// TIA Portal V20 export
DATA_BLOCK "InstCallEquipment"   // DB126
{ DB_Accessible_From_OPC_UA := 'FALSE' }
AUTHOR : ERsystem_FA2_DH. Kim
// stored: AssignedProDiagFB Unit1.Em3.ProDiag, DBAccessibleFromOPCUA false, DBAccessibleFromWebserver false, InstanceOfName Unit1.Em3.CallEquipment, InstanceOfType FB, Namespace Unit1.Em3
"Unit1.Em3.CallEquipment"
   // VAR_INPUT
   //    ZoneOperationEnable { ExternalWritable := 'False'} : "LWONIK_typeSafetyZoneManualOperation";
   // END_VAR
   // VAR_IN_OUT
   //    unitStatus : "LAF_typeUnitStatus";
   //    unitAlarmDB : "LAF_typeAlarms";
   //    emFeedback : "LUC_typeEmFeedback";
   // END_VAR
   // VAR
   //    InstSequenceWebGuide : "Unit1.Em3.Sequence_1_WebGuide";
   //    instWebGuideHomeJob1 { S7_SetPoint := 'True'} : "LAF_SelectJob";
   //    instWebGuideGuidingJob2 { S7_SetPoint := 'True'} : "LAF_SelectJob";
   //    instCmSafetyPinIdlePositionSensor : "LBC_DigitalSignalCn";
   //    instCmIonizerTopMaintDetection { S7_SetPoint := 'True'} : "LBC_DigitalSignalCn";
   //    instCmIonizerTopErrorDetection { S7_SetPoint := 'True'} : "LBC_DigitalSignalCn";
   //    instCmIonizerBtmMaintDetection { S7_SetPoint := 'True'} : "LBC_DigitalSignalCn";
   //    instCmIonizerBtmErrorDetection { S7_SetPoint := 'True'} : "LBC_DigitalSignalCn";
   //    instCmDancerEncoder { ExternalAccessible := 'False'; ExternalVisible := 'False'; ExternalWritable := 'False'; S7_SetPoint := 'True'} : "LBC_AnalogInputCn";
   //    instCmLoadCellControllerInterface { ExternalAccessible := 'False'; ExternalVisible := 'False'; ExternalWritable := 'False'; S7_SetPoint := 'True'} : "LBC_AnalogInputCn";
   //    instCmDancerElectroPneumaticRegulator { ExternalAccessible := 'False'; ExternalVisible := 'False'; ExternalWritable := 'False'; S7_SetPoint := 'True'} : "LBC_AnalogOutputCn";
   //    instCmCompensatorAxisX { S7_SetPoint := 'True'} : "LBC_Axis64Pos_TecPlcCn";
   //    instCmUnwinderVirtualAxisX { S7_SetPoint := 'True'} : "LBC_Axis64Pos_TecPlcCn";
   //    instInterlockCompensatorAxisX { S7_SetPoint := 'True'} : "LER_Axis64Pos_InterlockSummary";
   //    instInterlockUnwinderVirtualAxisX { S7_SetPoint := 'True'} : "LER_Axis64Pos_InterlockSummary";
   //    instCmDancerFwdBwd { ExternalAccessible := 'False'; ExternalVisible := 'False'; ExternalWritable := 'False'; S7_SetPoint := 'True'} : "LBC_TwoWayActuatorCn";
   //    instCmSepaUnwinderIonizerTop { ExternalAccessible := 'False'; ExternalVisible := 'False'; ExternalWritable := 'False'; S7_SetPoint := 'True'} : "LBC_TwoWayActuatorCn";
   //    instCmSepaUnwinderIonizerBottom { ExternalAccessible := 'False'; ExternalVisible := 'False'; ExternalWritable := 'False'; S7_SetPoint := 'True'} : "LBC_TwoWayActuatorCn";
   //    instCmEpcPivot { ExternalAccessible := 'False'; ExternalVisible := 'False'; ExternalWritable := 'False'; S7_SetPoint := 'True'} : "LER_EPC_CON600";
   //    instManageAlarms { ExternalWritable := 'False'} : "LAF_ManageAlarms";
   //    instEventsPFE : "Unit1.Em3.EventsPFE";
   //    statUnitStatus { ExternalWritable := 'False'} : "LAF_typeUnitStatus";
   //    statSlmStatus : Struct
   //       running { ExternalWritable := 'False'} : Bool;
   //       powerOff { ExternalWritable := 'False'} : Bool;
   //    END_STRUCT;
   //    statTonTime { ExternalAccessible := 'False'; ExternalVisible := 'False'; ExternalWritable := 'False'} : Array[0..1999] of TON_TIME;
   //    statTofTime { ExternalAccessible := 'False'; ExternalVisible := 'False'; ExternalWritable := 'False'} : Array[0..99] of TOF_TIME;
   //    statPulse { ExternalAccessible := 'False'; ExternalVisible := 'False'; ExternalWritable := 'False'} : Struct
   //       miscellaneous : Array[0..99] of Bool;
   //       workingDone : Struct
   //          mainPnP : Array[0..99] of Bool;
   //          alignTable : Array[0..99] of Bool;
   //          ngPnP : Array[0..99] of Bool;
   //       END_STRUCT;
   //       axisEnable : Array[0..99] of Bool;
   //       brakeTest : Array[0..99] of Bool;
   //    END_STRUCT;
   //    statEnableManualCmds : Bool := TRUE;
   //    Scan_on : Bool;
   //    "*** Interlock Axis ***" { ExternalAccessible := 'False'; ExternalVisible := 'False'; ExternalWritable := 'False'} : Bool;
   //    "compenastor X Home" { S7_SetPoint := 'True'} : "Homing.LER_Axis";
   //    "compenastor X Jog_CW" { S7_SetPoint := 'True'} : "Jog.LER_Axis";
   //    "compenastor X Jog_CCW" { S7_SetPoint := 'True'} : "Jog.LER_Axis";
   //    "compenastor X Position_" { S7_SetPoint := 'True'} : Array[0..5] of "Position.LER_Axis";
   //    "*** Interlock Actuator ******" { ExternalAccessible := 'False'; ExternalVisible := 'False'; ExternalWritable := 'False'} : Bool;
   //    "DancerFwdBwd Home" { S7_SetPoint := 'True'} : "Cylinder.LER_Actuator";
   //    "DancerFwdBwd Work" { S7_SetPoint := 'True'} : "Cylinder.LER_Actuator";
   //    "SepaUnwinderIonizer Home" { S7_SetPoint := 'True'} : "Cylinder.LER_Actuator";
   //    "SepaUnwinderIonizer Work" { S7_SetPoint := 'True'} : "Cylinder.LER_Actuator";
   //    "SepaUnwinderIonizerBottom Home" { S7_SetPoint := 'True'} : "Cylinder.LER_Actuator";
   //    "SepaUnwinderIonizerBottom Work" { S7_SetPoint := 'True'} : "Cylinder.LER_Actuator";
   //    AXIS3 : "LER_CM_Name";
   //    Cylinder10 : "LER_CM_Name";
   //    instCmRotaionSafetyPinPositionSensor { ExternalAccessible := 'False'; ExternalVisible := 'False'; ExternalWritable := 'False'} : "LBC_DigitalSignalCn";
   //    citi_Ptrig : Array[0..20] of Bool;
   //    citiTon : Array[0..20] of TON_TIME;
   //    citi : Time;
   //    citiTest : Array[0..20] of Bool;
   // END_VAR
BEGIN
   ZoneOperationEnable.autoStartEnable := FALSE;
   ZoneOperationEnable.doorLockEnable := TRUE;
   ZoneOperationEnable.doorUnlockEnable := TRUE;
   ZoneOperationEnable.rc_AutoEnable := FALSE;
   ZoneOperationEnable.rc_RollChangeEnable := FALSE;
   ZoneOperationEnable.rc_DoorLockEnable := TRUE;
   ZoneOperationEnable.rc_DoorUnlockEnable := TRUE;
   ZoneOperationEnable.hmiOperationEnable := TRUE;
   ZoneOperationEnable.phmiOperationEnable := FALSE;
   instCmSafetyPinIdlePositionSensor.enable := TRUE;
   instCmSafetyPinIdlePositionSensor.parentReferenceDesignator := WSTRING#'U1.EM3 WebGuide';
   instCmSafetyPinIdlePositionSensor.digitalValue := TRUE;
   instCmSafetyPinIdlePositionSensor.simulatedDigitalValue := FALSE;
   instCmSafetyPinIdlePositionSensor.statProcessValues.enable := TRUE;
   instCmSafetyPinIdlePositionSensor.statProcessValues.referenceDesignator := WSTRING#'U1.EM3 WebGuide.DigitalSignal';
   instCmSafetyPinIdlePositionSensor.statProcessValues.simulation := FALSE;
   instCmSafetyPinIdlePositionSensor.statProcessValues.processValue := TRUE;
   instCmSafetyPinIdlePositionSensor.statProcessValues.error := FALSE;
   instCmSafetyPinIdlePositionSensor.statProcessValues.status := 16#0000;
   instCmSafetyPinIdlePositionSensor.statDiagnostics.status := 16#0000;
   instCmSafetyPinIdlePositionSensor.statDiagnostics.subfunctionStatus := 16#0000;
   instCmSafetyPinIdlePositionSensor.statDiagnostics.stateNumber := 0;
   instCmSafetyPinIdlePositionSensor.statEmptyDiagnostics.status := 16#0000;
   instCmSafetyPinIdlePositionSensor.statEmptyDiagnostics.subfunctionStatus := 16#0000;
   instCmSafetyPinIdlePositionSensor.statEmptyDiagnostics.stateNumber := 0;
   instCmSafetyPinIdlePositionSensor.instOnDelay.PT := T#0MS;
   instCmSafetyPinIdlePositionSensor.instOnDelay.IN := FALSE;
   instCmSafetyPinIdlePositionSensor.instOffDelay.PT := T#0MS;
   instCmSafetyPinIdlePositionSensor.instOffDelay.IN := FALSE;
   instCmSafetyPinIdlePositionSensor.statDisableAlarms := FALSE;
   instCmSafetyPinIdlePositionSensor.statErrorState := 16#0000;
   instCmSafetyPinIdlePositionSensor.statFirstCall := FALSE;
   instCmSafetyPinIdlePositionSensor.statResetPrevious := FALSE;
   instCmSafetyPinIdlePositionSensor.statEnablePrevious := TRUE;
   instCmSafetyPinIdlePositionSensor.statProcessValuePrevious := TRUE;
   instCmIonizerTopMaintDetection.enable := TRUE;
   instCmIonizerTopMaintDetection.parentReferenceDesignator := WSTRING#'U1.EM3 WebGuide';
   instCmIonizerTopMaintDetection.digitalValue := FALSE;
   instCmIonizerTopMaintDetection.simulatedDigitalValue := FALSE;
   instCmIonizerTopMaintDetection.statProcessValues.enable := TRUE;
   instCmIonizerTopMaintDetection.statProcessValues.referenceDesignator := WSTRING#'U1.EM3 WebGuide.DigitalSignal';
   instCmIonizerTopMaintDetection.statProcessValues.simulation := FALSE;
   instCmIonizerTopMaintDetection.statProcessValues.processValue := FALSE;
   instCmIonizerTopMaintDetection.statProcessValues.error := FALSE;
   instCmIonizerTopMaintDetection.statProcessValues.status := 16#0000;
   instCmIonizerTopMaintDetection.statDiagnostics.status := 16#0000;
   instCmIonizerTopMaintDetection.statDiagnostics.subfunctionStatus := 16#0000;
   instCmIonizerTopMaintDetection.statDiagnostics.stateNumber := 0;
   instCmIonizerTopMaintDetection.statEmptyDiagnostics.status := 16#0000;
   instCmIonizerTopMaintDetection.statEmptyDiagnostics.subfunctionStatus := 16#0000;
   instCmIonizerTopMaintDetection.statEmptyDiagnostics.stateNumber := 0;
   instCmIonizerTopMaintDetection.instOnDelay.PT := T#0MS;
   instCmIonizerTopMaintDetection.instOnDelay.IN := FALSE;
   instCmIonizerTopMaintDetection.instOffDelay.PT := T#0MS;
   instCmIonizerTopMaintDetection.instOffDelay.IN := FALSE;
   instCmIonizerTopMaintDetection.statDisableAlarms := FALSE;
   instCmIonizerTopMaintDetection.statErrorState := 16#0000;
   instCmIonizerTopMaintDetection.statFirstCall := FALSE;
   instCmIonizerTopMaintDetection.statResetPrevious := FALSE;
   instCmIonizerTopMaintDetection.statEnablePrevious := TRUE;
   instCmIonizerTopMaintDetection.statProcessValuePrevious := FALSE;
   instCmIonizerTopErrorDetection.enable := TRUE;
   instCmIonizerTopErrorDetection.parentReferenceDesignator := WSTRING#'U1.EM3 WebGuide';
   instCmIonizerTopErrorDetection.digitalValue := TRUE;
   instCmIonizerTopErrorDetection.simulatedDigitalValue := FALSE;
   instCmIonizerTopErrorDetection.statProcessValues.enable := TRUE;
   instCmIonizerTopErrorDetection.statProcessValues.referenceDesignator := WSTRING#'U1.EM3 WebGuide.DigitalSignal';
   instCmIonizerTopErrorDetection.statProcessValues.simulation := FALSE;
   instCmIonizerTopErrorDetection.statProcessValues.processValue := TRUE;
   instCmIonizerTopErrorDetection.statProcessValues.error := FALSE;
   instCmIonizerTopErrorDetection.statProcessValues.status := 16#0000;
   instCmIonizerTopErrorDetection.statDiagnostics.status := 16#0000;
   instCmIonizerTopErrorDetection.statDiagnostics.subfunctionStatus := 16#0000;
   instCmIonizerTopErrorDetection.statDiagnostics.stateNumber := 0;
   instCmIonizerTopErrorDetection.statEmptyDiagnostics.status := 16#0000;
   instCmIonizerTopErrorDetection.statEmptyDiagnostics.subfunctionStatus := 16#0000;
   instCmIonizerTopErrorDetection.statEmptyDiagnostics.stateNumber := 0;
   instCmIonizerTopErrorDetection.instOnDelay.PT := T#0MS;
   instCmIonizerTopErrorDetection.instOnDelay.IN := FALSE;
   instCmIonizerTopErrorDetection.instOffDelay.PT := T#0MS;
   instCmIonizerTopErrorDetection.instOffDelay.IN := FALSE;
   instCmIonizerTopErrorDetection.statDisableAlarms := FALSE;
   instCmIonizerTopErrorDetection.statErrorState := 16#0000;
   instCmIonizerTopErrorDetection.statFirstCall := FALSE;
   instCmIonizerTopErrorDetection.statResetPrevious := FALSE;
   instCmIonizerTopErrorDetection.statEnablePrevious := TRUE;
   instCmIonizerTopErrorDetection.statProcessValuePrevious := TRUE;
   instCmIonizerBtmMaintDetection.enable := TRUE;
   instCmIonizerBtmMaintDetection.parentReferenceDesignator := WSTRING#'U1.EM3 WebGuide';
   instCmIonizerBtmMaintDetection.digitalValue := FALSE;
   instCmIonizerBtmMaintDetection.simulatedDigitalValue := FALSE;
   instCmIonizerBtmMaintDetection.statProcessValues.enable := TRUE;
   instCmIonizerBtmMaintDetection.statProcessValues.referenceDesignator := WSTRING#'U1.EM3 WebGuide.DigitalSignal';
   instCmIonizerBtmMaintDetection.statProcessValues.simulation := FALSE;
   instCmIonizerBtmMaintDetection.statProcessValues.processValue := FALSE;
   instCmIonizerBtmMaintDetection.statProcessValues.error := FALSE;
   instCmIonizerBtmMaintDetection.statProcessValues.status := 16#0000;
   instCmIonizerBtmMaintDetection.statDiagnostics.status := 16#0000;
   instCmIonizerBtmMaintDetection.statDiagnostics.subfunctionStatus := 16#0000;
   instCmIonizerBtmMaintDetection.statDiagnostics.stateNumber := 0;
   instCmIonizerBtmMaintDetection.statEmptyDiagnostics.status := 16#0000;
   instCmIonizerBtmMaintDetection.statEmptyDiagnostics.subfunctionStatus := 16#0000;
   instCmIonizerBtmMaintDetection.statEmptyDiagnostics.stateNumber := 0;
   instCmIonizerBtmMaintDetection.instOnDelay.PT := T#0MS;
   instCmIonizerBtmMaintDetection.instOnDelay.IN := FALSE;
   instCmIonizerBtmMaintDetection.instOffDelay.PT := T#0MS;
   instCmIonizerBtmMaintDetection.instOffDelay.IN := FALSE;
   instCmIonizerBtmMaintDetection.statDisableAlarms := FALSE;
   instCmIonizerBtmMaintDetection.statErrorState := 16#0000;
   instCmIonizerBtmMaintDetection.statFirstCall := FALSE;
   instCmIonizerBtmMaintDetection.statResetPrevious := FALSE;
   instCmIonizerBtmMaintDetection.statEnablePrevious := TRUE;
   instCmIonizerBtmMaintDetection.statProcessValuePrevious := FALSE;
   instCmIonizerBtmErrorDetection.enable := TRUE;
   instCmIonizerBtmErrorDetection.parentReferenceDesignator := WSTRING#'U1.EM3 WebGuide';
   instCmIonizerBtmErrorDetection.digitalValue := TRUE;
   instCmIonizerBtmErrorDetection.simulatedDigitalValue := FALSE;
   instCmIonizerBtmErrorDetection.statProcessValues.enable := TRUE;
   instCmIonizerBtmErrorDetection.statProcessValues.referenceDesignator := WSTRING#'U1.EM3 WebGuide.DigitalSignal';
   instCmIonizerBtmErrorDetection.statProcessValues.simulation := FALSE;
   instCmIonizerBtmErrorDetection.statProcessValues.processValue := TRUE;
   instCmIonizerBtmErrorDetection.statProcessValues.error := FALSE;
   instCmIonizerBtmErrorDetection.statProcessValues.status := 16#0000;
   instCmIonizerBtmErrorDetection.statDiagnostics.status := 16#0000;
   instCmIonizerBtmErrorDetection.statDiagnostics.subfunctionStatus := 16#0000;
   instCmIonizerBtmErrorDetection.statDiagnostics.stateNumber := 0;
   instCmIonizerBtmErrorDetection.statEmptyDiagnostics.status := 16#0000;
   instCmIonizerBtmErrorDetection.statEmptyDiagnostics.subfunctionStatus := 16#0000;
   instCmIonizerBtmErrorDetection.statEmptyDiagnostics.stateNumber := 0;
   instCmIonizerBtmErrorDetection.instOnDelay.PT := T#0MS;
   instCmIonizerBtmErrorDetection.instOnDelay.IN := FALSE;
   instCmIonizerBtmErrorDetection.instOffDelay.PT := T#0MS;
   instCmIonizerBtmErrorDetection.instOffDelay.IN := FALSE;
   instCmIonizerBtmErrorDetection.statDisableAlarms := FALSE;
   instCmIonizerBtmErrorDetection.statErrorState := 16#0000;
   instCmIonizerBtmErrorDetection.statFirstCall := FALSE;
   instCmIonizerBtmErrorDetection.statResetPrevious := FALSE;
   instCmIonizerBtmErrorDetection.statEnablePrevious := TRUE;
   instCmIonizerBtmErrorDetection.statProcessValuePrevious := TRUE;
   instCmDancerEncoder.enable := TRUE;
   instCmDancerEncoder.parentReferenceDesignator := WSTRING#'U1.EM3 WebGuide';
   instCmDancerEncoder.analogValue := 13938;
   instCmDancerEncoder.simulatedAnalogValue := 0;
   instCmDancerEncoder.statProcessValues.enable := TRUE;
   instCmDancerEncoder.statProcessValues.referenceDesignator := WSTRING#'U1.EM3 WebGuide.cmDancerEncoder';
   instCmDancerEncoder.statProcessValues.simulation := FALSE;
   instCmDancerEncoder.statProcessValues.processValue := 0.354600694444443;
   instCmDancerEncoder.statProcessValues.analogValue := 13879;
   instCmDancerEncoder.statProcessValues.limitHigh2 := FALSE;
   instCmDancerEncoder.statProcessValues.limitHigh1 := FALSE;
   instCmDancerEncoder.statProcessValues.limitLow1 := FALSE;
   instCmDancerEncoder.statProcessValues.limitLow2 := FALSE;
   instCmDancerEncoder.statProcessValues.maxValueReached := FALSE;
   instCmDancerEncoder.statProcessValues.minValueReached := FALSE;
   instCmDancerEncoder.statProcessValues.error := FALSE;
   instCmDancerEncoder.statProcessValues.status := 16#0000;
   instCmDancerEncoder.statDiagnostics.status := 16#0000;
   instCmDancerEncoder.statDiagnostics.subfunctionStatus := 16#0000;
   instCmDancerEncoder.statDiagnostics.stateNumber := 0;
   instCmDancerEncoder.statEmptyDiagnostics.status := 16#0000;
   instCmDancerEncoder.statEmptyDiagnostics.subfunctionStatus := 16#0000;
   instCmDancerEncoder.statEmptyDiagnostics.stateNumber := 0;
   instCmDancerEncoder.statLimitationMessage := '';
   instCmDancerEncoder.statLimitMessage := '';
   instCmDancerEncoder.statErrorState := 16#0000;
   instCmDancerEncoder.statFirstCall := FALSE;
   instCmDancerEncoder.statDisableAlarms := FALSE;
   instCmDancerEncoder.statResetPrevious := FALSE;
   instCmDancerEncoder.statEnablePrevious := TRUE;
   instCmLoadCellControllerInterface.enable := TRUE;
   instCmLoadCellControllerInterface.parentReferenceDesignator := WSTRING#'U1.EM3 WebGuide';
   instCmLoadCellControllerInterface.analogValue := 5;
   instCmLoadCellControllerInterface.simulatedAnalogValue := 0;
   instCmLoadCellControllerInterface.statProcessValues.enable := TRUE;
   instCmLoadCellControllerInterface.statProcessValues.referenceDesignator := WSTRING#'U1.EM3 WebGuide.cmLoadCellController';
   instCmLoadCellControllerInterface.statProcessValues.simulation := FALSE;
   instCmLoadCellControllerInterface.statProcessValues.processValue := -99.9638310185185;
   instCmLoadCellControllerInterface.statProcessValues.analogValue := 5;
   instCmLoadCellControllerInterface.statProcessValues.limitHigh2 := FALSE;
   instCmLoadCellControllerInterface.statProcessValues.limitHigh1 := FALSE;
   instCmLoadCellControllerInterface.statProcessValues.limitLow1 := TRUE;
   instCmLoadCellControllerInterface.statProcessValues.limitLow2 := TRUE;
   instCmLoadCellControllerInterface.statProcessValues.maxValueReached := FALSE;
   instCmLoadCellControllerInterface.statProcessValues.minValueReached := FALSE;
   instCmLoadCellControllerInterface.statProcessValues.error := FALSE;
   instCmLoadCellControllerInterface.statProcessValues.status := 16#0000;
   instCmLoadCellControllerInterface.statDiagnostics.status := 16#0000;
   instCmLoadCellControllerInterface.statDiagnostics.subfunctionStatus := 16#0000;
   instCmLoadCellControllerInterface.statDiagnostics.stateNumber := 0;
   instCmLoadCellControllerInterface.statEmptyDiagnostics.status := 16#0000;
   instCmLoadCellControllerInterface.statEmptyDiagnostics.subfunctionStatus := 16#0000;
   instCmLoadCellControllerInterface.statEmptyDiagnostics.stateNumber := 0;
   instCmLoadCellControllerInterface.statLimitationMessage := '';
   instCmLoadCellControllerInterface.statLimitMessage := '-99.96 unit <= -90.00 unit';
   instCmLoadCellControllerInterface.statErrorState := 16#0000;
   instCmLoadCellControllerInterface.statFirstCall := FALSE;
   instCmLoadCellControllerInterface.statDisableAlarms := TRUE;
   instCmLoadCellControllerInterface.statResetPrevious := FALSE;
   instCmLoadCellControllerInterface.statEnablePrevious := TRUE;
   instCmDancerElectroPneumaticRegulator.enable := TRUE;
   instCmDancerElectroPneumaticRegulator.parentReferenceDesignator := WSTRING#'';
   instCmDancerElectroPneumaticRegulator.processValue := 0.0;
   instCmDancerElectroPneumaticRegulator.simulatedProcessValue := 0.0;
   instCmDancerElectroPneumaticRegulator.analogValue := 0;
   instCmDancerElectroPneumaticRegulator.statProcessValues.enable := TRUE;
   instCmDancerElectroPneumaticRegulator.statProcessValues.referenceDesignator := WSTRING#'cmDancerRegulator';
   instCmDancerElectroPneumaticRegulator.statProcessValues.simulation := FALSE;
   instCmDancerElectroPneumaticRegulator.statProcessValues.processValue := 0.0;
   instCmDancerElectroPneumaticRegulator.statProcessValues.analogValue := 0;
   instCmDancerElectroPneumaticRegulator.statProcessValues.limitHigh2 := FALSE;
   instCmDancerElectroPneumaticRegulator.statProcessValues.limitHigh1 := FALSE;
   instCmDancerElectroPneumaticRegulator.statProcessValues.limitLow1 := TRUE;
   instCmDancerElectroPneumaticRegulator.statProcessValues.limitLow2 := TRUE;
   instCmDancerElectroPneumaticRegulator.statProcessValues.maxValueReached := FALSE;
   instCmDancerElectroPneumaticRegulator.statProcessValues.minValueReached := FALSE;
   instCmDancerElectroPneumaticRegulator.statProcessValues.error := FALSE;
   instCmDancerElectroPneumaticRegulator.statProcessValues.status := 16#0000;
   instCmDancerElectroPneumaticRegulator.statDiagnostics.status := 16#0000;
   instCmDancerElectroPneumaticRegulator.statDiagnostics.subfunctionStatus := 16#0000;
   instCmDancerElectroPneumaticRegulator.statDiagnostics.stateNumber := 0;
   instCmDancerElectroPneumaticRegulator.statEmptyDiagnostics.status := 16#0000;
   instCmDancerElectroPneumaticRegulator.statEmptyDiagnostics.subfunctionStatus := 16#0000;
   instCmDancerElectroPneumaticRegulator.statEmptyDiagnostics.stateNumber := 0;
   instCmDancerElectroPneumaticRegulator.statLimitationMessage := '';
   instCmDancerElectroPneumaticRegulator.statLimitMessage := '0.00 unit <= 0.00 unit';
   instCmDancerElectroPneumaticRegulator.statErrorState := 16#0000;
   instCmDancerElectroPneumaticRegulator.statFirstCall := FALSE;
   instCmDancerElectroPneumaticRegulator.statDisableAlarms := TRUE;
   instCmDancerElectroPneumaticRegulator.statResetPrevious := FALSE;
   instCmDancerElectroPneumaticRegulator.statEnablePrevious := TRUE;
   instCmDancerFwdBwd.enable := TRUE;
   instCmDancerFwdBwd.parentReferenceDesignator := WSTRING#'U1.EM3 WebGuide';
   instCmDancerFwdBwd.feedbackHomePos := FALSE;
   instCmDancerFwdBwd.feedbackWorkPos := FALSE;
   instCmDancerFwdBwd.enableManualCmds := TRUE;
   instCmDancerFwdBwd.interlockWorkPos := TRUE;
   instCmDancerFwdBwd.interlockHomePos := TRUE;
   instCmDancerFwdBwd.goToHomePos := FALSE;
   instCmDancerFwdBwd.goToWorkPos := FALSE;
   instCmDancerFwdBwd.statProcessValues.enable := TRUE;
   instCmDancerFwdBwd.statProcessValues.referenceDesignator := WSTRING#'U1.EM3 WebGuide.cmDancerFwdBwd';
   instCmDancerFwdBwd.statProcessValues.commandHomePos := FALSE;
   instCmDancerFwdBwd.statProcessValues.commandWorkPos := FALSE;
   instCmDancerFwdBwd.statProcessValues.goToHomePos := FALSE;
   instCmDancerFwdBwd.statProcessValues.goToWorkPos := FALSE;
   instCmDancerFwdBwd.statProcessValues.inHomePos := FALSE;
   instCmDancerFwdBwd.statProcessValues.inWorkPos := FALSE;
   instCmDancerFwdBwd.statProcessValues.reset := FALSE;
   instCmDancerFwdBwd.statProcessValues.enableManualCmds := TRUE;
   instCmDancerFwdBwd.statProcessValues.error := FALSE;
   instCmDancerFwdBwd.statProcessValues.interlockHomePos := TRUE;
   instCmDancerFwdBwd.statProcessValues.interlockWorkPos := TRUE;
   instCmDancerFwdBwd.statProcessValues.status := 16#7003;
   instCmDancerFwdBwd.statProcessValues.interlockWarningWorkPos := FALSE;
   instCmDancerFwdBwd.statProcessValues.interlockWarningHomePos := FALSE;
   instCmDancerFwdBwd.statCurrentInputs.commandHomePos := FALSE;
   instCmDancerFwdBwd.statCurrentInputs.commandWorkPos := FALSE;
   instCmDancerFwdBwd.statCurrentInputs.reset := FALSE;
   instCmDancerFwdBwd.statPreviousInputs.commandHomePos := FALSE;
   instCmDancerFwdBwd.statPreviousInputs.commandWorkPos := FALSE;
   instCmDancerFwdBwd.statPreviousInputs.reset := FALSE;
   instCmDancerFwdBwd.statCurrentInterface.commandHomePos := FALSE;
   instCmDancerFwdBwd.statCurrentInterface.commandWorkPos := FALSE;
   instCmDancerFwdBwd.statCurrentInterface.reset := FALSE;
   instCmDancerFwdBwd.statPreviousInterface.commandHomePos := FALSE;
   instCmDancerFwdBwd.statPreviousInterface.commandWorkPos := FALSE;
   instCmDancerFwdBwd.statPreviousInterface.reset := FALSE;
   instCmDancerFwdBwd.statEmptyDiagnostics.status := 16#0000;
   instCmDancerFwdBwd.statEmptyDiagnostics.subfunctionStatus := 16#0000;
   instCmDancerFwdBwd.statEmptyDiagnostics.stateNumber := 0;
   instCmDancerFwdBwd.instTimerReachPos.PT := T#0MS;
   instCmDancerFwdBwd.instTimerReachPos.IN := FALSE;
   instCmDancerFwdBwd.instTimerLeavePos.PT := T#0MS;
   instCmDancerFwdBwd.instTimerLeavePos.IN := FALSE;
   instCmDancerFwdBwd.instTimerDiscrepancyCheck.PT := T#0MS;
   instCmDancerFwdBwd.instTimerDiscrepancyCheck.IN := FALSE;
   instCmDancerFwdBwd.statDisableAlarms := TRUE;
   instCmDancerFwdBwd.statDiagnostics.status := 16#7003;
   instCmDancerFwdBwd.statDiagnostics.subfunctionStatus := 16#0000;
   instCmDancerFwdBwd.statDiagnostics.stateNumber := 0;
   instCmDancerFwdBwd.statEnablePrevious := TRUE;
   instCmDancerFwdBwd.statFirstCall := FALSE;
   instCmDancerFwdBwd.statResetPrevious := FALSE;
   instCmDancerFwdBwd.statValid := TRUE;
   instCmDancerFwdBwd.statBusy := TRUE;
   instCmDancerFwdBwd.statError := FALSE;
   instCmDancerFwdBwd.statInterlockWorkOff := FALSE;
   instCmDancerFwdBwd.statInterlockHomeOff := FALSE;
   instCmDancerFwdBwd.statFbState := 50;
   instCmDancerFwdBwd.statFbStatePrevious := 50;
   instCmDancerFwdBwd.statErrorUserCleared := FALSE;
   instCmDancerFwdBwd.statErrorAutoCleared := FALSE;
   instCmDancerFwdBwd.statErrorState := 16#0000;
   instCmDancerFwdBwd.statDisablingCompleted := FALSE;
   instCmDancerFwdBwd.statFeedbackHomePos := FALSE;
   instCmDancerFwdBwd.statFeedbackWorkPos := FALSE;
   instCmSepaUnwinderIonizerTop.enable := TRUE;
   instCmSepaUnwinderIonizerTop.parentReferenceDesignator := WSTRING#'U1.EM3 WebGuide';
   instCmSepaUnwinderIonizerTop.feedbackHomePos := FALSE;
   instCmSepaUnwinderIonizerTop.feedbackWorkPos := FALSE;
   instCmSepaUnwinderIonizerTop.enableManualCmds := TRUE;
   instCmSepaUnwinderIonizerTop.interlockWorkPos := TRUE;
   instCmSepaUnwinderIonizerTop.interlockHomePos := TRUE;
   instCmSepaUnwinderIonizerTop.goToHomePos := FALSE;
   instCmSepaUnwinderIonizerTop.goToWorkPos := FALSE;
   instCmSepaUnwinderIonizerTop.statProcessValues.enable := TRUE;
   instCmSepaUnwinderIonizerTop.statProcessValues.referenceDesignator := WSTRING#'U1.EM3 WebGuide.cmSepaUnwinderIonizerTop';
   instCmSepaUnwinderIonizerTop.statProcessValues.commandHomePos := FALSE;
   instCmSepaUnwinderIonizerTop.statProcessValues.commandWorkPos := FALSE;
   instCmSepaUnwinderIonizerTop.statProcessValues.goToHomePos := FALSE;
   instCmSepaUnwinderIonizerTop.statProcessValues.goToWorkPos := FALSE;
   instCmSepaUnwinderIonizerTop.statProcessValues.inHomePos := FALSE;
   instCmSepaUnwinderIonizerTop.statProcessValues.inWorkPos := FALSE;
   instCmSepaUnwinderIonizerTop.statProcessValues.reset := FALSE;
   instCmSepaUnwinderIonizerTop.statProcessValues.enableManualCmds := TRUE;
   instCmSepaUnwinderIonizerTop.statProcessValues.error := FALSE;
   instCmSepaUnwinderIonizerTop.statProcessValues.interlockHomePos := TRUE;
   instCmSepaUnwinderIonizerTop.statProcessValues.interlockWorkPos := TRUE;
   instCmSepaUnwinderIonizerTop.statProcessValues.status := 16#7003;
   instCmSepaUnwinderIonizerTop.statProcessValues.interlockWarningWorkPos := FALSE;
   instCmSepaUnwinderIonizerTop.statProcessValues.interlockWarningHomePos := FALSE;
   instCmSepaUnwinderIonizerTop.statCurrentInputs.commandHomePos := FALSE;
   instCmSepaUnwinderIonizerTop.statCurrentInputs.commandWorkPos := FALSE;
   instCmSepaUnwinderIonizerTop.statCurrentInputs.reset := FALSE;
   instCmSepaUnwinderIonizerTop.statPreviousInputs.commandHomePos := FALSE;
   instCmSepaUnwinderIonizerTop.statPreviousInputs.commandWorkPos := FALSE;
   instCmSepaUnwinderIonizerTop.statPreviousInputs.reset := FALSE;
   instCmSepaUnwinderIonizerTop.statCurrentInterface.commandHomePos := FALSE;
   instCmSepaUnwinderIonizerTop.statCurrentInterface.commandWorkPos := FALSE;
   instCmSepaUnwinderIonizerTop.statCurrentInterface.reset := FALSE;
   instCmSepaUnwinderIonizerTop.statPreviousInterface.commandHomePos := FALSE;
   instCmSepaUnwinderIonizerTop.statPreviousInterface.commandWorkPos := FALSE;
   instCmSepaUnwinderIonizerTop.statPreviousInterface.reset := FALSE;
   instCmSepaUnwinderIonizerTop.statEmptyDiagnostics.status := 16#0000;
   instCmSepaUnwinderIonizerTop.statEmptyDiagnostics.subfunctionStatus := 16#0000;
   instCmSepaUnwinderIonizerTop.statEmptyDiagnostics.stateNumber := 0;
   instCmSepaUnwinderIonizerTop.instTimerReachPos.PT := T#0MS;
   instCmSepaUnwinderIonizerTop.instTimerReachPos.IN := FALSE;
   instCmSepaUnwinderIonizerTop.instTimerLeavePos.PT := T#0MS;
   instCmSepaUnwinderIonizerTop.instTimerLeavePos.IN := FALSE;
   instCmSepaUnwinderIonizerTop.instTimerDiscrepancyCheck.PT := T#0MS;
   instCmSepaUnwinderIonizerTop.instTimerDiscrepancyCheck.IN := FALSE;
   instCmSepaUnwinderIonizerTop.statDisableAlarms := FALSE;
   instCmSepaUnwinderIonizerTop.statDiagnostics.status := 16#7003;
   instCmSepaUnwinderIonizerTop.statDiagnostics.subfunctionStatus := 16#0000;
   instCmSepaUnwinderIonizerTop.statDiagnostics.stateNumber := 0;
   instCmSepaUnwinderIonizerTop.statEnablePrevious := TRUE;
   instCmSepaUnwinderIonizerTop.statFirstCall := FALSE;
   instCmSepaUnwinderIonizerTop.statResetPrevious := FALSE;
   instCmSepaUnwinderIonizerTop.statValid := TRUE;
   instCmSepaUnwinderIonizerTop.statBusy := TRUE;
   instCmSepaUnwinderIonizerTop.statError := FALSE;
   instCmSepaUnwinderIonizerTop.statInterlockWorkOff := FALSE;
   instCmSepaUnwinderIonizerTop.statInterlockHomeOff := FALSE;
   instCmSepaUnwinderIonizerTop.statFbState := 50;
   instCmSepaUnwinderIonizerTop.statFbStatePrevious := 50;
   instCmSepaUnwinderIonizerTop.statErrorUserCleared := FALSE;
   instCmSepaUnwinderIonizerTop.statErrorAutoCleared := FALSE;
   instCmSepaUnwinderIonizerTop.statErrorState := 16#0000;
   instCmSepaUnwinderIonizerTop.statDisablingCompleted := FALSE;
   instCmSepaUnwinderIonizerTop.statFeedbackHomePos := FALSE;
   instCmSepaUnwinderIonizerTop.statFeedbackWorkPos := FALSE;
   instCmSepaUnwinderIonizerBottom.enable := TRUE;
   instCmSepaUnwinderIonizerBottom.parentReferenceDesignator := WSTRING#'U1.EM3 WebGuide';
   instCmSepaUnwinderIonizerBottom.feedbackHomePos := FALSE;
   instCmSepaUnwinderIonizerBottom.feedbackWorkPos := FALSE;
   instCmSepaUnwinderIonizerBottom.enableManualCmds := TRUE;
   instCmSepaUnwinderIonizerBottom.interlockWorkPos := TRUE;
   instCmSepaUnwinderIonizerBottom.interlockHomePos := TRUE;
   instCmSepaUnwinderIonizerBottom.goToHomePos := FALSE;
   instCmSepaUnwinderIonizerBottom.goToWorkPos := FALSE;
   instCmSepaUnwinderIonizerBottom.statProcessValues.enable := TRUE;
   instCmSepaUnwinderIonizerBottom.statProcessValues.referenceDesignator := WSTRING#'U1.EM3 WebGuide.cmSepaUnwinderIonizerBtm';
   instCmSepaUnwinderIonizerBottom.statProcessValues.commandHomePos := FALSE;
   instCmSepaUnwinderIonizerBottom.statProcessValues.commandWorkPos := FALSE;
   instCmSepaUnwinderIonizerBottom.statProcessValues.goToHomePos := FALSE;
   instCmSepaUnwinderIonizerBottom.statProcessValues.goToWorkPos := FALSE;
   instCmSepaUnwinderIonizerBottom.statProcessValues.inHomePos := FALSE;
   instCmSepaUnwinderIonizerBottom.statProcessValues.inWorkPos := FALSE;
   instCmSepaUnwinderIonizerBottom.statProcessValues.reset := FALSE;
   instCmSepaUnwinderIonizerBottom.statProcessValues.enableManualCmds := TRUE;
   instCmSepaUnwinderIonizerBottom.statProcessValues.error := FALSE;
   instCmSepaUnwinderIonizerBottom.statProcessValues.interlockHomePos := TRUE;
   instCmSepaUnwinderIonizerBottom.statProcessValues.interlockWorkPos := TRUE;
   instCmSepaUnwinderIonizerBottom.statProcessValues.status := 16#7003;
   instCmSepaUnwinderIonizerBottom.statProcessValues.interlockWarningWorkPos := FALSE;
   instCmSepaUnwinderIonizerBottom.statProcessValues.interlockWarningHomePos := FALSE;
   instCmSepaUnwinderIonizerBottom.statCurrentInputs.commandHomePos := FALSE;
   instCmSepaUnwinderIonizerBottom.statCurrentInputs.commandWorkPos := FALSE;
   instCmSepaUnwinderIonizerBottom.statCurrentInputs.reset := FALSE;
   instCmSepaUnwinderIonizerBottom.statPreviousInputs.commandHomePos := FALSE;
   instCmSepaUnwinderIonizerBottom.statPreviousInputs.commandWorkPos := FALSE;
   instCmSepaUnwinderIonizerBottom.statPreviousInputs.reset := FALSE;
   instCmSepaUnwinderIonizerBottom.statCurrentInterface.commandHomePos := FALSE;
   instCmSepaUnwinderIonizerBottom.statCurrentInterface.commandWorkPos := FALSE;
   instCmSepaUnwinderIonizerBottom.statCurrentInterface.reset := FALSE;
   instCmSepaUnwinderIonizerBottom.statPreviousInterface.commandHomePos := FALSE;
   instCmSepaUnwinderIonizerBottom.statPreviousInterface.commandWorkPos := FALSE;
   instCmSepaUnwinderIonizerBottom.statPreviousInterface.reset := FALSE;
   instCmSepaUnwinderIonizerBottom.statEmptyDiagnostics.status := 16#0000;
   instCmSepaUnwinderIonizerBottom.statEmptyDiagnostics.subfunctionStatus := 16#0000;
   instCmSepaUnwinderIonizerBottom.statEmptyDiagnostics.stateNumber := 0;
   instCmSepaUnwinderIonizerBottom.instTimerReachPos.PT := T#0MS;
   instCmSepaUnwinderIonizerBottom.instTimerReachPos.IN := FALSE;
   instCmSepaUnwinderIonizerBottom.instTimerLeavePos.PT := T#0MS;
   instCmSepaUnwinderIonizerBottom.instTimerLeavePos.IN := FALSE;
   instCmSepaUnwinderIonizerBottom.instTimerDiscrepancyCheck.PT := T#0MS;
   instCmSepaUnwinderIonizerBottom.instTimerDiscrepancyCheck.IN := FALSE;
   instCmSepaUnwinderIonizerBottom.statDisableAlarms := FALSE;
   instCmSepaUnwinderIonizerBottom.statDiagnostics.status := 16#7003;
   instCmSepaUnwinderIonizerBottom.statDiagnostics.subfunctionStatus := 16#0000;
   instCmSepaUnwinderIonizerBottom.statDiagnostics.stateNumber := 0;
   instCmSepaUnwinderIonizerBottom.statEnablePrevious := TRUE;
   instCmSepaUnwinderIonizerBottom.statFirstCall := FALSE;
   instCmSepaUnwinderIonizerBottom.statResetPrevious := FALSE;
   instCmSepaUnwinderIonizerBottom.statValid := TRUE;
   instCmSepaUnwinderIonizerBottom.statBusy := TRUE;
   instCmSepaUnwinderIonizerBottom.statError := FALSE;
   instCmSepaUnwinderIonizerBottom.statInterlockWorkOff := FALSE;
   instCmSepaUnwinderIonizerBottom.statInterlockHomeOff := FALSE;
   instCmSepaUnwinderIonizerBottom.statFbState := 50;
   instCmSepaUnwinderIonizerBottom.statFbStatePrevious := 50;
   instCmSepaUnwinderIonizerBottom.statErrorUserCleared := FALSE;
   instCmSepaUnwinderIonizerBottom.statErrorAutoCleared := FALSE;
   instCmSepaUnwinderIonizerBottom.statErrorState := 16#0000;
   instCmSepaUnwinderIonizerBottom.statDisablingCompleted := FALSE;
   instCmSepaUnwinderIonizerBottom.statFeedbackHomePos := FALSE;
   instCmSepaUnwinderIonizerBottom.statFeedbackWorkPos := FALSE;
   instManageAlarms.proDiagState.Total_Number := 459;
   instManageAlarms.proDiagState.All := TRUE;
   instManageAlarms.proDiagState.O := FALSE;
   instManageAlarms.proDiagState.I := FALSE;
   instManageAlarms.proDiagState.R := FALSE;
   instManageAlarms.proDiagState."A" := FALSE;
   instManageAlarms.proDiagState.P := FALSE;
   instManageAlarms.proDiagState.Merr := TRUE;
   instManageAlarms.proDiagState.Mtxt := FALSE;
   instManageAlarms.proDiagState.SV_Types := 16#20;
   instManageAlarms.proDiagState.C1 := TRUE;
   instManageAlarms.proDiagState.C2 := FALSE;
   instManageAlarms.proDiagState.C3 := FALSE;
   instManageAlarms.proDiagState.C4 := FALSE;
   instManageAlarms.proDiagState.C5 := FALSE;
   instManageAlarms.proDiagState.C6 := FALSE;
   instManageAlarms.proDiagState.C7 := FALSE;
   instManageAlarms.proDiagState.C8 := FALSE;
   instManageAlarms.proDiagState.Categories := 16#01;
   instManageAlarms.proDiagState.Sub_Cat_1 := 16#0000_0001;
   instManageAlarms.proDiagState.Sub_Cat_2 := 16#0000_0000;
   instManageAlarms.proDiagState.Reserved := 16#00;
   instManageAlarms.parentAlarmDB.error := TRUE;
   instManageAlarms.parentAlarmDB.warning := FALSE;
   instManageAlarms.parentAlarmDB.info := FALSE;
   instManageAlarms.alarmDB.error := TRUE;
   instManageAlarms.alarmDB.warning := FALSE;
   instManageAlarms.alarmDB.info := FALSE;
   instManageAlarms.hmiInterfaceDB.error := TRUE;
   instManageAlarms.hmiInterfaceDB.warning := FALSE;
   instManageAlarms.hmiInterfaceDB.info := FALSE;
   statUnitStatus.acknowledgeActive := FALSE;
   statUnitStatus.alarmsDisabled := FALSE;
   statUnitStatus.simulationActive := FALSE;
   statUnitStatus.safetyReleased := TRUE;
   statUnitStatus.specialFunctions.GaugeRnR1AnodeAlign := FALSE;
   statUnitStatus.specialFunctions.GaugeRnR1CathodeAlign := FALSE;
   statUnitStatus.specialFunctions.GaugeRnR3AnodeAlign := FALSE;
   statUnitStatus.specialFunctions.GaugeRnR3CathodeAlign := FALSE;
   statUnitStatus.specialFunctions.releaseEntry := FALSE;
   statUnitStatus.specialFunctions.dryRun := FALSE;
   statUnitStatus.specialFunctions.ReelCutAnodeUnuse := FALSE;
   statUnitStatus.mode.current := 2;
   statUnitStatus.mode.production := FALSE;
   statUnitStatus.mode.maintenance := TRUE;
   statUnitStatus.mode.manual := FALSE;
   statUnitStatus.mode.sleep := FALSE;
   statUnitStatus.mode.deepsleep := FALSE;
   statUnitStatus.mode.userMode04 := FALSE;
   statUnitStatus.mode.userMode05 := FALSE;
   statUnitStatus.mode.userMode06 := FALSE;
   statUnitStatus.mode.userMode07 := FALSE;
   statUnitStatus.mode.userMode08 := FALSE;
   statUnitStatus.mode.userMode09 := FALSE;
   statUnitStatus.mode.userMode10 := FALSE;
   statUnitStatus.mode.userMode11 := FALSE;
   statUnitStatus.mode.userMode12 := FALSE;
   statUnitStatus.mode.userMode13 := FALSE;
   statUnitStatus.state.current := 2;
   statUnitStatus.state.clearing := FALSE;
   statUnitStatus.state.stopped := TRUE;
   statUnitStatus.state.starting := FALSE;
   statUnitStatus.state.idle := FALSE;
   statUnitStatus.state.suspended := FALSE;
   statUnitStatus.state.execute := FALSE;
   statUnitStatus.state.stopping := FALSE;
   statUnitStatus.state.aborting := FALSE;
   statUnitStatus.state.aborted := FALSE;
   statUnitStatus.state.holding := FALSE;
   statUnitStatus.state.held := FALSE;
   statUnitStatus.state.unholding := FALSE;
   statUnitStatus.state.suspending := FALSE;
   statUnitStatus.state.unsuspending := FALSE;
   statUnitStatus.state.resetting := FALSE;
   statUnitStatus.state.completing := FALSE;
   statUnitStatus.state.complete := FALSE;
END_DATA_BLOCK
